{attribute 'qualified_only'}
{attribute 'strict'}
TYPE eCoolingControl :
(
	off := 0,
	temporary := 1,
	full := 2
);
END_TYPE

(* stored: Version 1.1.0.1, ProductVersion 3.1.4024.12
   DUT eCoolingControl: Id {7ef18c95-c231-49cd-b5c2-587d96a85996} *)
